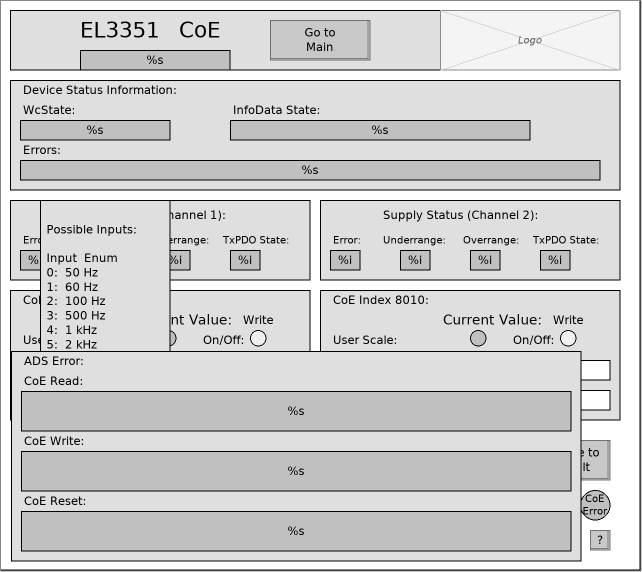
VISUALIZATION VISU_EL3351_CoE  // 642x572
VAR_IN_OUT
	m_Input_afbEL3351_Index_ : FB_EL3351;
END_VAR
    Rectangle (0,0 640x570)
    Rectangle (10,10 610x60)
    Rectangle (70,10 100x40), "EL3351"
    Image (440,10 180x60), image: Logo
    Image (440,10 180x60), image: Logo
    Rectangle (150,10 100x40), "CoE"
    Button (270,20 100x40), "Go to Main"
        p3450524324: m_Input_afbEL3351_Index_.dwButtonColour
        tap m_Input_afbEL3351_Index_.bCoEZoom
    Rectangle (10,200 300x80)
    Rectangle (20,230 50x20), "Error:"
    Rectangle (320,200 300x80)
    Rectangle (220,230 110x20), "TxPDO State:"
    Rectangle (150,230 90x20), "Overrange:"
    Rectangle (70,230 100x20), "Underrange:"
    Rectangle (330,230 50x20), "Error:"
    Rectangle (380,230 100x20), "Underrange:"
    Rectangle (460,230 90x20), "Overrange:"
    Rectangle (530,230 110x20), "TxPDO State:"
    Rectangle (320,290 300x130)
    Ellipse (470,330 16x16), colour variable: m_Input_afbEL3351_Index_.fbCoe.dwUserScaleReadIndex8010
    RoundedRectangle (440,360 80x20), "%d", text variable: m_Input_afbEL3351_Index_.fbCoE.astCoeRead[6].nData, colour variable: m_Input_afbEL3351_Index_.fbCoe.dwUserScaleOffsetReadIndex8010
    RoundedRectangle (440,390 80x20), "%d", text variable: m_Input_afbEL3351_Index_.fbCoE.astCoeRead[7].nData, colour variable: m_Input_afbEL3351_Index_.fbCoe.dwUserScaleGainReadIndex8010
    Rectangle (330,290 120x20), "CoE Index 8010:"
    Rectangle (550,310 50x20), "Write"
    Ellipse (560,330 16x16), colour variable: m_Input_afbEL3351_Index_.fbCoe.dwUserScaleWriteIndex8010
        toggle m_Input_afbEL3351_Index_.fbCoE.stCoe.bEnableUserScaleIndex8010
    RoundedRectangle (530,360 80x20), "%d", text variable: m_Input_afbEL3351_Index_.fbCoE.stCoe.diUserScaleOffsetIndex8010, input disabled if: NOT m_Input_afbEL3351_Index_.fbcoe.stCoe.bEnableUserScaleIndex8010, colour variable: m_Input_afbEL3351_Index_.fbCoe.dwUserScaleOffsetWriteIndex8010
        OnMouseDown: write the text variable via Edit
    RoundedRectangle (530,390 80x20), "%d", text variable: m_Input_afbEL3351_Index_.fbCoE.stCoe.diUserScaleGainIndex8010, input disabled if: NOT m_Input_afbEL3351_Index_.fbcoe.stCoe.bEnableUserScaleIndex8010, colour variable: m_Input_afbEL3351_Index_.fbCoe.dwUserScaleGainWriteIndex8010
        OnMouseDown: write the text variable via Edit
    Rectangle (330,330 90x20), "User Scale:"
    Rectangle (330,360 130x20), "User Scale Offset:"
    Rectangle (330,390 130x20), "User Scale Gain:"
    Rectangle (440,310 100x20), "Current Value:"
    Rectangle (10,290 300x130)
    Rectangle (20,330 90x20), "User Scale:"
    Ellipse (160,330 16x16), colour variable: m_Input_afbEL3351_Index_.fbCoe.dwUserScaleRead
    Rectangle (20,360 130x20), "User Scale Offset:"
    Rectangle (20,390 130x20), "User Scale Gain:"
    RoundedRectangle (130,360 80x20), "%d", text variable: m_Input_afbEL3351_Index_.fbCoE.astCoeRead[2].nData, colour variable: m_Input_afbEL3351_Index_.fbCoe.dwUserScaleOffsetRead
    RoundedRectangle (130,390 80x20), "%d", text variable: m_Input_afbEL3351_Index_.fbCoE.astCoeRead[3].nData, colour variable: m_Input_afbEL3351_Index_.fbCoe.dwUserScaleGainRead
    Rectangle (20,290 130x20), "CoE Index 8000:"
    RoundedRectangle (220,360 80x20), "%d", text variable: m_Input_afbEL3351_Index_.fbCoE.stCoe.diUserScaleOffset, input disabled if: NOT m_Input_afbEL3351_Index_.fbcoe.stCoe.bEnableUserScale, colour variable: m_Input_afbEL3351_Index_.fbCoe.dwUserScaleOffsetWrite
        OnMouseDown: write the text variable via Edit
    RoundedRectangle (220,390 80x20), "%d", text variable: m_Input_afbEL3351_Index_.fbCoE.stCoe.diUserScaleGain, input disabled if: NOT m_Input_afbEL3351_Index_.fbcoe.stCoe.bEnableUserScale, colour variable: m_Input_afbEL3351_Index_.fbCoe.dwUserScaleGainWrite
        OnMouseDown: write the text variable via Edit
    Rectangle (130,310 100x20), "Current Value:"
    Rectangle (240,310 50x20), "Write"
    Ellipse (250,330 16x16), colour variable: m_Input_afbEL3351_Index_.fbCoe.dwUserScaleWrite
        toggle m_Input_afbEL3351_Index_.fbCoE.stCoe.bEnableUserScale
    Rectangle (200,330 50x20), "On/Off:"
    Rectangle (510,330 50x20), "On/Off:"
    Rectangle (70,200 190x30), "Bridge Status (Channel 1):"
    Rectangle (380,200 180x30), "Supply Status (Channel 2):"
    RoundedRectangle (20,250 30x20), "%i", text variable: m_Input_afbEL3351_Index_.fbChannelDiagnosis.bBridgeError, colour variable: m_Input_afbEL3351_Index_.fbChannelDiagnosis.dwBridgeErrorColour
    RoundedRectangle (90,250 30x20), "%i", text variable: m_Input_afbEL3351_Index_.fbChannelDiagnosis.bBridgeUnderrange, colour variable: m_Input_afbEL3351_Index_.fbChannelDiagnosis.dwBridgeUnderrangeColour
    RoundedRectangle (160,250 30x20), "%i", text variable: m_Input_afbEL3351_Index_.fbChannelDiagnosis.bBridgeOverrangerange, colour variable: m_Input_afbEL3351_Index_.fbChannelDiagnosis.dwBridgeOverrangerangeColour
    RoundedRectangle (230,250 30x20), "%i", text variable: m_Input_afbEL3351_Index_.fbChannelDiagnosis.bBridgeState, colour variable: m_Input_afbEL3351_Index_.fbChannelDiagnosis.dwBridgeStateColour
    RoundedRectangle (330,250 30x20), "%i", text variable: m_Input_afbEL3351_Index_.fbChannelDiagnosis.bSupplyError, colour variable: m_Input_afbEL3351_Index_.fbChannelDiagnosis.dwSupplyErrorColour
    RoundedRectangle (400,250 30x20), "%i", text variable: m_Input_afbEL3351_Index_.fbChannelDiagnosis.bSupplyUnderrange, colour variable: m_Input_afbEL3351_Index_.fbChannelDiagnosis.dwSupplyUnderrangeColour
    RoundedRectangle (470,250 30x20), "%i", text variable: m_Input_afbEL3351_Index_.fbChannelDiagnosis.bSupplyOverrangerange, colour variable: m_Input_afbEL3351_Index_.fbChannelDiagnosis.dwSupplyOverrangerangeColour
    RoundedRectangle (540,250 30x20), "%i", text variable: m_Input_afbEL3351_Index_.fbChannelDiagnosis.bSupplyState, colour variable: m_Input_afbEL3351_Index_.fbChannelDiagnosis.dwSupplyStateColour
    Polygon (620,430)
    Rectangle (20,530 110x20), "Update Time:"
    RoundedRectangle (160,530 60x20), "%.4f s", text variable: m_Input_afbEL3351_Index_.fbToggleBit.rUpdateTime
    Rectangle (20,500 140x20), "Toggle Bit Counter:"
    RoundedRectangle (160,500 60x20), "%.0f", text variable: m_Input_afbEL3351_Index_.fbToggleBit.rToggleBitCounter
    RoundedRectangle (240,470 70x20), "%s", text variable: m_Input_afbEL3351_Index_.fbCoE.sFilterSettings
    Rectangle (250,450 60x20), "Enum:"
    RoundedRectangle (160,470 60x20), "%d", text variable: m_Input_afbEL3351_Index_.fbCoE.stCoe.dwFilterSettings, colour variable: m_Input_afbEL3351_Index_.fbCoe.dwFilterWrite
        OnMouseDown: write the text variable via Edit
    RoundedRectangle (80,470 60x20), "%d", text variable: m_Input_afbEL3351_Index_.fbCoE.astCoeRead[4].nData, colour variable: m_Input_afbEL3351_Index_.fbCoe.dwFilterRead
    Rectangle (20,430 100x30), "Filter:"
    Rectangle (170,450 50x20), "Write"
    Rectangle (70,450 100x20), "Current Value:"
    Button (130,520 20x20), "?", pressed state: m_Input_afbEL3351_Index_.bQuestionMarkToggle
        p3450524324: m_Input_afbEL3351_Index_.dwButtonColour
        toggle m_Input_afbEL3351_Index_.bQuestionMarkToggle
    Button (20,460 20x20), "?", pressed state: m_Input_afbEL3351_Index_.bQuestionMarkFilter
        p3450524324: m_Input_afbEL3351_Index_.dwButtonColour
        toggle m_Input_afbEL3351_Index_.bQuestionMarkFilter
    Rectangle (330,500 200x20), "%s", text variable: m_Input_afbEL3351_Index_.fbCoE.sStatus
    Ellipse (580,490 30x30), "CoE Error", colour toggle: (m_Input_afbEL3351_Index_.fbCoE.bCoeError) <> 0
    Button (530,440 80x40), "Set Coe to default"
        p3450524324: m_Input_afbEL3351_Index_.dwButtonColour
        tap m_Input_afbEL3351_Index_.fbCoE.bButtonSetCoeParametersToDefault
    Button (430,440 80x40), "Write CoE"
        p3450524324: m_Input_afbEL3351_Index_.fbCoe.dwWriteColour
        tap m_Input_afbEL3351_Index_.fbCoE.bButtonWriteCoeParameters
    Button (330,440 80x40), "Read CoE"
        p3450524324: m_Input_afbEL3351_Index_.dwButtonColour
        tap m_Input_afbEL3351_Index_.fbCoE.bButtonReadCoeParameters
    Rectangle (40,200 130x260), "Possible Inputs: Input Enum 0: 50 Hz 1: 60 Hz 2: 100 Hz 3: 500 Hz 4: 1 kHz 5: 2 kHz 6: 3.75 kHz 7: 7.5 kHz 8: 15 kHz 9: 30 kHz 10: 5 Hz 11: 10 Hz", invisible if: NOT m_Input_afbEL3351_Index_.bQuestionMarkFilter
    Rectangle (250,530 330x20), "%s", text variable: m_Input_afbEL3351_Index_.fbCoE.sStatusCoeAccess, colour variable: m_Input_afbEL3351_Index_.fbCoe.dwStatusCoeAccess
    Rectangle (40,440 290x80), "For a period of 10 seconds, it is checked how often the Toggle Bit is set. Then, the update time is calculated: Update Time = 1/ (Toggle Bit / 10)", invisible if: NOT m_Input_afbEL3351_Index_.bQuestionMarkToggle
    Ellipse (540,490 30x30), "CoE Busy", colour toggle: (m_Input_afbEL3351_Index_.fbCoE.bCoeBusy) <> 0
    Button (590,530 20x20), "?", pressed state: m_Input_afbEL3351_Index_.bQuestionMarkAdsError
        p3450524324: m_Input_afbEL3351_Index_.dwButtonColour
        toggle m_Input_afbEL3351_Index_.bQuestionMarkAdsError
    Group (11,351 568x208), invisible if: NOT m_Input_afbEL3351_Index_.bQuestionMarkAdsError
        Rectangle (0,0 570x210)
        Rectangle (10,0 210x20), "ADS Error:"
        Rectangle (10,160 550x40), "%s", text variable: m_Input_afbEL3351_Index_.fbCoe.sAdsErrorTextReset, colour variable: m_Input_afbEL3351_Index_.fbCoe.dwCoeErrorTextReset
        Rectangle (10,40 550x40), "%s", text variable: m_Input_afbEL3351_Index_.fbCoe.sAdsErrorTextRead, colour variable: m_Input_afbEL3351_Index_.fbCoe.dwCoeErrorTextRead
        Rectangle (10,100 550x40), "%s", text variable: m_Input_afbEL3351_Index_.fbCoe.sAdsErrorTextWrite, colour variable: m_Input_afbEL3351_Index_.fbCoe.dwCoeErrorTextWrite
        Rectangle (10,20 90x20), "CoE Read:"
        Rectangle (10,140 100x20), "CoE Reset:"
        Rectangle (10,80 90x20), "CoE Write:"
    Rectangle (10,80 610x110)
    Rectangle (20,80 190x20), "Device Status Information:"
    Rectangle (230,120 300x20), "%s", text variable: m_Input_afbEL3351_Index_.fbTerminalDiagnosis.sState, colour variable: m_Input_afbEL3351_Index_.fbTerminalDiagnosis.dwStateStatusColour
    Rectangle (20,120 150x20), "%s", text variable: m_Input_afbEL3351_Index_.fbTerminalDiagnosis.sWorkingState, colour variable: m_Input_afbEL3351_Index_.fbTerminalDiagnosis.dwWcStateColour
    Rectangle (20,160 580x20), "%s", text variable: m_Input_afbEL3351_Index_.fbTerminalDiagnosis.sStateStatusAll, colour variable: m_Input_afbEL3351_Index_.fbTerminalDiagnosis.dwStateStatusAllColour
    Rectangle (20,100 90x20), "WcState:"
    Rectangle (230,100 120x20), "InfoData State:"
    Rectangle (20,140 70x20), "Errors:"
    Rectangle (80,50 150x20), "%s", text variable: m_Input_afbEL3351_Index_.sShowTerminalNumber
END_VISUALIZATION

(* stored: Version 1.1.0.1, ProductVersion 3.1.4024.12
   Visu VISU_EL3351_CoE: Id {34603a37-1c94-4cde-97ff-744ef54abc60} *)
